FUNCTION_BLOCK FB_SVs_Ablaufsteuerung
VAR_IN_OUT
	Zustand			: ST_SVs_Zustand;
	Stellwert		: ST_SV_Stellwert;
END_VAR
VAR_INPUT
	Steuerung		: ST_SV_Steuerung;
	Parameter		: ST_SV_Parameter;
END_VAR
VAR_OUTPUT
END_VAR
VAR
END_VAR

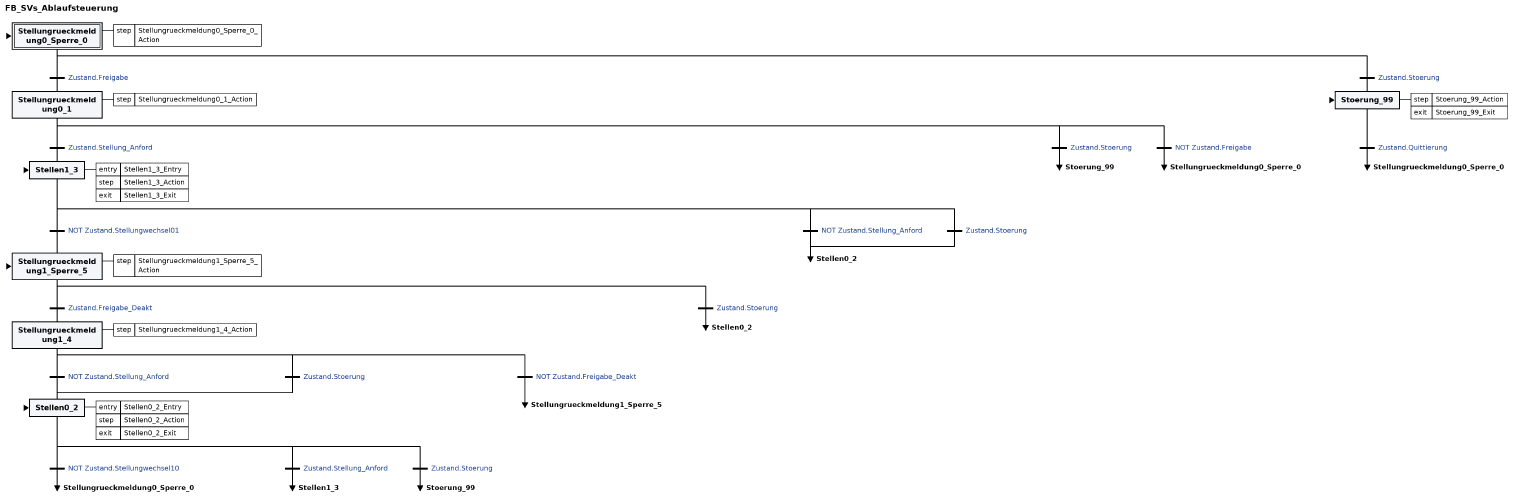
INITIAL_STEP Stellungrueckmeldung0_Sperre_0:
    Stellungrueckmeldung0_Sperre_0_Action(N);  // step action
END_STEP
TRANSITION FROM Stellungrueckmeldung0_Sperre_0 TO Stellungrueckmeldung0_1
    := Zustand.Freigabe;
END_TRANSITION
TRANSITION FROM Stellungrueckmeldung0_Sperre_0 TO Stoerung_99
    := Zustand.Stoerung;
END_TRANSITION
STEP Stoerung_99:
    Stoerung_99_Action(N);  // step action
    Stoerung_99_Exit(P0);  // exit action
END_STEP
TRANSITION FROM Stoerung_99 TO Stellungrueckmeldung0_Sperre_0
    := Zustand.Quittierung;
END_TRANSITION
STEP Stellungrueckmeldung0_1:
    Stellungrueckmeldung0_1_Action(N);  // step action
END_STEP
TRANSITION FROM Stellungrueckmeldung0_1 TO Stellen1_3
    := Zustand.Stellung_Anford;
END_TRANSITION
TRANSITION FROM Stellungrueckmeldung0_1 TO Stoerung_99
    := Zustand.Stoerung;
END_TRANSITION
TRANSITION FROM Stellungrueckmeldung0_1 TO Stellungrueckmeldung0_Sperre_0
    := NOT Zustand.Freigabe;
END_TRANSITION
STEP Stellen1_3:
    Stellen1_3_Entry(P1);  // entry action
    Stellen1_3_Action(N);  // step action
    Stellen1_3_Exit(P0);  // exit action
END_STEP
TRANSITION FROM Stellen1_3 TO Stellungrueckmeldung1_Sperre_5
    := NOT Zustand.Stellungwechsel01;
END_TRANSITION
TRANSITION FROM Stellen1_3 TO Stellen0_2
    := NOT Zustand.Stellung_Anford;
END_TRANSITION
TRANSITION FROM Stellen1_3 TO Stellen0_2
    := Zustand.Stoerung;
END_TRANSITION
STEP Stellungrueckmeldung1_Sperre_5:
    Stellungrueckmeldung1_Sperre_5_Action(N);  // step action
END_STEP
TRANSITION FROM Stellungrueckmeldung1_Sperre_5 TO Stellungrueckmeldung1_4
    := Zustand.Freigabe_Deakt;
END_TRANSITION
TRANSITION FROM Stellungrueckmeldung1_Sperre_5 TO Stellen0_2
    := Zustand.Stoerung;
END_TRANSITION
STEP Stellungrueckmeldung1_4:
    Stellungrueckmeldung1_4_Action(N);  // step action
END_STEP
TRANSITION FROM Stellungrueckmeldung1_4 TO Stellen0_2
    := NOT Zustand.Stellung_Anford;
END_TRANSITION
TRANSITION FROM Stellungrueckmeldung1_4 TO Stellen0_2
    := Zustand.Stoerung;
END_TRANSITION
TRANSITION FROM Stellungrueckmeldung1_4 TO Stellungrueckmeldung1_Sperre_5
    := NOT Zustand.Freigabe_Deakt;
END_TRANSITION
STEP Stellen0_2:
    Stellen0_2_Entry(P1);  // entry action
    Stellen0_2_Action(N);  // step action
    Stellen0_2_Exit(P0);  // exit action
END_STEP
TRANSITION FROM Stellen0_2 TO Stellungrueckmeldung0_Sperre_0
    := NOT Zustand.Stellungwechsel10;
END_TRANSITION
TRANSITION FROM Stellen0_2 TO Stellen1_3
    := Zustand.Stellung_Anford;
END_TRANSITION
TRANSITION FROM Stellen0_2 TO Stoerung_99
    := Zustand.Stoerung;
END_TRANSITION

ACTION Stellen0_2_Action:
(* Stellwert setzen *)
Stellwert.Stellung := FALSE;

(* Zustand setzen *)
Zustand.Stellungwechsel10 := NOT (Zustand.Stellungrueckmeldung0 AND (NOT Zustand.Stellungrueckmeldung1)) ;
Zustand.Status := E_Stellventil_Zustand_Stellungwechsel10;
END_ACTION

ACTION Stellen0_2_Entry:
Zustand.Stellungwechsel10 := TRUE;
END_ACTION

ACTION Stellen0_2_Exit:
Zustand.Stellungwechsel10 := FALSE;
END_ACTION

ACTION Stellen1_3_Action:
(* Stellwert setzen *)
Stellwert.Stellung := TRUE;

(* Zustand setzen *)
Zustand.Stellungwechsel01 := NOT(Zustand.Stellungrueckmeldung1 AND (NOT Zustand.Stellungrueckmeldung0));
Zustand.Status := E_Stellventil_Zustand_Stellungwechsel01;
END_ACTION

ACTION Stellen1_3_Entry:
Zustand.Stellungwechsel01 := TRUE;
END_ACTION

ACTION Stellen1_3_Exit:
Zustand.Stellungwechsel01 := FALSE;
END_ACTION

ACTION Stellungrueckmeldung0_1_Action:
(* Stellwert setzen *)
Stellwert.Stellung := FALSE;
Zustand.Stellung := FALSE;

(* Zustand setzen *)
Zustand.Status := E_Stellventil_Zustand_Status_Stellungrueckmeldung0;
END_ACTION

ACTION Stellungrueckmeldung0_Sperre_0_Action:
(* Stellwert setzen *)
Stellwert.Stellung := FALSE;
Zustand.Stellung := FALSE;

(* Zustand setzen *)
Zustand.Status := E_Stellventil_Zustand_Status_Stellungrueckmeldung0_Sperre;
END_ACTION

ACTION Stellungrueckmeldung1_4_Action:
(* Stellwert setzen *)
Stellwert.Stellung := TRUE;
Zustand.Stellung := TRUE;

(* Zustand setzen *)
Zustand.Status := E_Stellventil_Zustand_Status_Stellungrueckmeldung1;
END_ACTION

ACTION Stellungrueckmeldung1_Sperre_5_Action:
(* Stellwert setzen *)
Stellwert.Stellung := TRUE;
Zustand.Stellung := TRUE;

(* Zustand setzen *)
Zustand.Status := E_Stellventil_Zustand_Status_Stellungrueckmeldung1_Sperre;
END_ACTION

ACTION Stoerung_99_Action:
(* Stellwert setzen *)
Stellwert.Stellung := Zustand.Stellung;

(* Zustand setzen *)
Zustand.Stoerung := TRUE;
Zustand.Status := E_PU_Zustand_Status_Stoerung;
END_ACTION

ACTION Stoerung_99_Exit:
Zustand.Stoerung	:= FALSE;
END_ACTION

END_FUNCTION_BLOCK

(* stored: Version 1.1.0.1, ProductVersion 3.1.4024.9
   POU FB_SVs_Ablaufsteuerung: Id {a8b4173e-aeb5-4ca6-bab1-43ba495afc35}, SpecialFunc None
   Action Stellen0_2_Action: Id {f1b6e63f-f160-4f59-9cdf-6322aa8a039c}
   Action Stellen0_2_Entry: Id {227f7e17-6fe6-473f-bb2c-45414e0d05f0}
   Action Stellen0_2_Exit: Id {84199a2c-85f2-422d-8c66-b1e0d44919b7}
   Action Stellen1_3_Action: Id {f034a278-f6a7-42e3-a5fb-75ed3dacc027}
   Action Stellen1_3_Entry: Id {b6502346-771e-4ddf-9b2f-bcb6cef3120c}
   Action Stellen1_3_Exit: Id {8a0e4381-b27e-4957-98de-a6eb4343bee0}
   Action Stellungrueckmeldung0_1_Action: Id {80db6d3c-9c61-439d-8da7-6ca66b15e26f}
   Action Stellungrueckmeldung0_Sperre_0_Action: Id {9d5c9f1d-09ec-47b5-afe7-71b03c01994f}
   Action Stellungrueckmeldung1_4_Action: Id {38807c81-0db2-4872-b631-ec9627a18239}
   Action Stellungrueckmeldung1_Sperre_5_Action: Id {acd124ad-30f2-494a-b1fb-2310daf726b3}
   Action Stoerung_99_Action: Id {b6106753-654f-4add-a9fb-713c291eebbb}
   Action Stoerung_99_Exit: Id {cebd515b-6081-45f9-bc26-b64ffadde523} *)
